PROGRAM Alarm_1
VAR
	Always_ON				:	BOOL	:=TRUE	;//상시 ON
	Always_OFF				:	BOOL	:=FALSE	;//상시 OFF
END_VAR

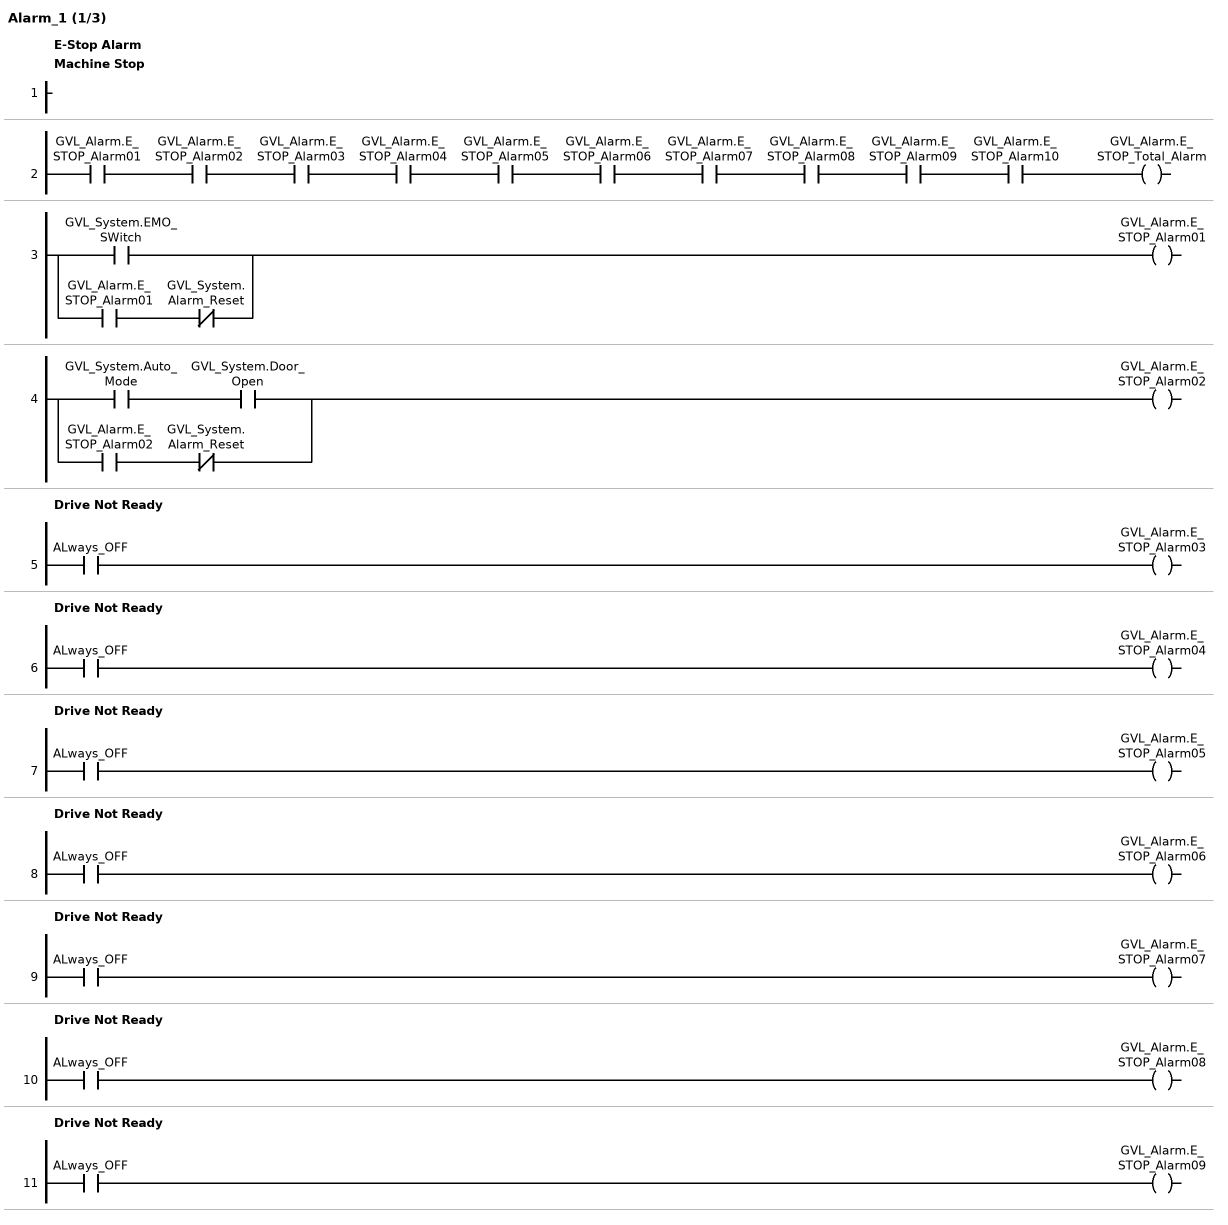
// NETWORK 1: E-Stop Alarm Machine Stop

// NETWORK 2
GVL_Alarm.E_STOP_Total_Alarm := GVL_Alarm.E_STOP_Alarm01 AND GVL_Alarm.E_STOP_Alarm02 AND GVL_Alarm.E_STOP_Alarm03 AND GVL_Alarm.E_STOP_Alarm04 AND GVL_Alarm.E_STOP_Alarm05 AND GVL_Alarm.E_STOP_Alarm06 AND GVL_Alarm.E_STOP_Alarm07 AND GVL_Alarm.E_STOP_Alarm08 AND GVL_Alarm.E_STOP_Alarm09 AND GVL_Alarm.E_STOP_Alarm10;

// NETWORK 3
GVL_Alarm.E_STOP_Alarm01 := GVL_System.EMO_SWitch OR GVL_Alarm.E_STOP_Alarm01 AND NOT GVL_System.Alarm_Reset;

// NETWORK 4
GVL_Alarm.E_STOP_Alarm02 := GVL_System.Auto_Mode AND GVL_System.Door_Open OR GVL_Alarm.E_STOP_Alarm02 AND NOT GVL_System.Alarm_Reset;

// NETWORK 5: Drive Not Ready
GVL_Alarm.E_STOP_Alarm03 := ALways_OFF;

// NETWORK 6: Drive Not Ready
GVL_Alarm.E_STOP_Alarm04 := ALways_OFF;

// NETWORK 7: Drive Not Ready
GVL_Alarm.E_STOP_Alarm05 := ALways_OFF;

// NETWORK 8: Drive Not Ready
GVL_Alarm.E_STOP_Alarm06 := ALways_OFF;

// NETWORK 9: Drive Not Ready
GVL_Alarm.E_STOP_Alarm07 := ALways_OFF;

// NETWORK 10: Drive Not Ready
GVL_Alarm.E_STOP_Alarm08 := ALways_OFF;

// NETWORK 11: Drive Not Ready
GVL_Alarm.E_STOP_Alarm09 := ALways_OFF;

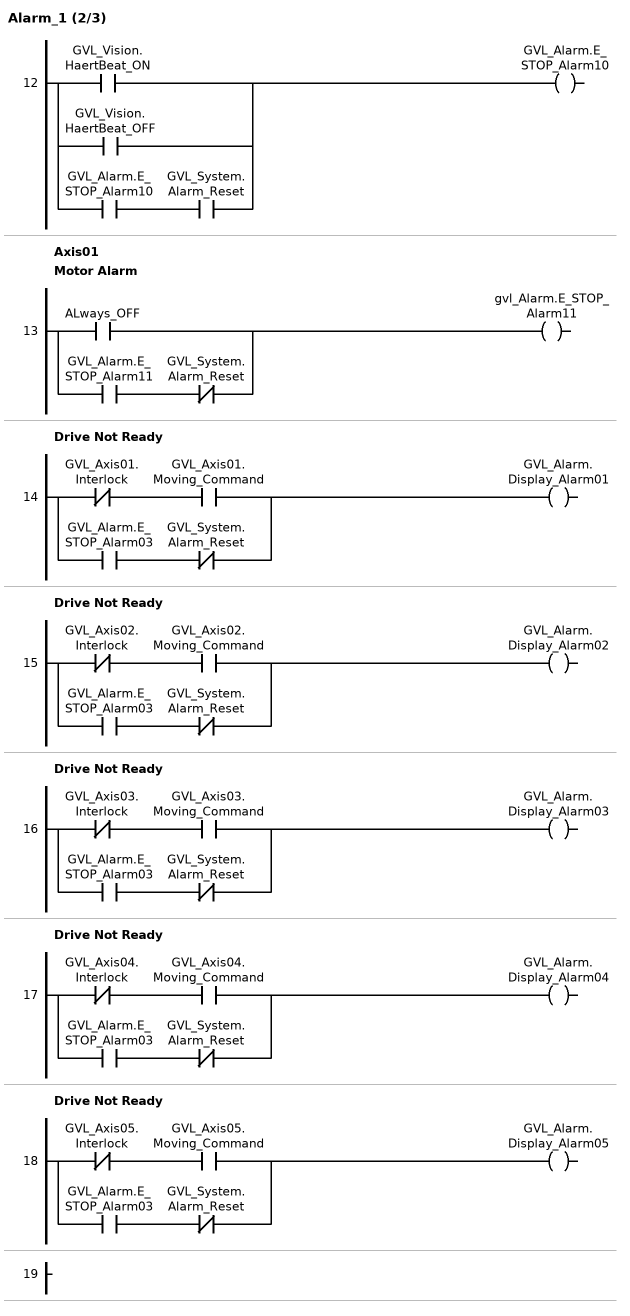
// NETWORK 12
GVL_Alarm.E_STOP_Alarm10 := GVL_Vision.HaertBeat_ON OR GVL_Vision.HaertBeat_OFF OR GVL_Alarm.E_STOP_Alarm10 AND GVL_System.Alarm_Reset;

// NETWORK 13: Axis01 Motor Alarm
gvl_Alarm.E_STOP_Alarm11 := ALways_OFF OR GVL_Alarm.E_STOP_Alarm11 AND NOT GVL_System.Alarm_Reset;

// NETWORK 14: Drive Not Ready
GVL_Alarm.Display_Alarm01 := NOT GVL_Axis01.Interlock AND GVL_Axis01.Moving_Command OR GVL_Alarm.E_STOP_Alarm03 AND NOT GVL_System.Alarm_Reset;

// NETWORK 15: Drive Not Ready
GVL_Alarm.Display_Alarm02 := NOT GVL_Axis02.Interlock AND GVL_Axis02.Moving_Command OR GVL_Alarm.E_STOP_Alarm03 AND NOT GVL_System.Alarm_Reset;

// NETWORK 16: Drive Not Ready
GVL_Alarm.Display_Alarm03 := NOT GVL_Axis03.Interlock AND GVL_Axis03.Moving_Command OR GVL_Alarm.E_STOP_Alarm03 AND NOT GVL_System.Alarm_Reset;

// NETWORK 17: Drive Not Ready
GVL_Alarm.Display_Alarm04 := NOT GVL_Axis04.Interlock AND GVL_Axis04.Moving_Command OR GVL_Alarm.E_STOP_Alarm03 AND NOT GVL_System.Alarm_Reset;

// NETWORK 18: Drive Not Ready
GVL_Alarm.Display_Alarm05 := NOT GVL_Axis05.Interlock AND GVL_Axis05.Moving_Command OR GVL_Alarm.E_STOP_Alarm03 AND NOT GVL_System.Alarm_Reset;

// NETWORK 19

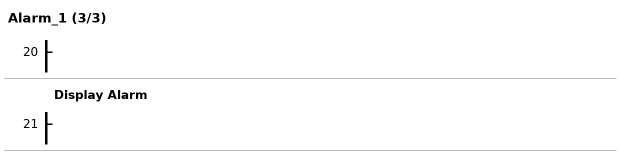
// NETWORK 20

// NETWORK 21: Display Alarm

END_PROGRAM

(* stored: Version 1.1.0.1, ProductVersion 3.1.4024.15
   POU Alarm_1: Id {02a7614f-d007-47e6-9563-898688ebd80e}, SpecialFunc None *)
